INTERFACE I_Module

METHOD Disable
VAR_INPUT
END_VAR
END_METHOD

METHOD Enable
VAR_INPUT
END_VAR
END_METHOD

END_INTERFACE

(* stored: Version 1.1.0.1, ProductVersion 3.1.4024.11
   Itf I_Module: Id {3db5525d-1ae8-43f9-a20d-7168266d3543}
   Method Disable: Id {c78a835b-990c-4da8-adea-19c0c0a74e46}
   Method Enable: Id {17ee0c27-8910-45cc-8c09-9f0461a06c75} *)
